(* PLC project Unnamed, Unknown Unnamed 1 *)
(* stored: creationDateTime 2024-07-23T15:43:19, modificationDateTime 2024-07-23T15:49:17 *)

PROGRAM program0
  VAR
    LocalVar0 : BOOL;
    LocalVar1 : SINT;
  END_VAR
  VAR  (* added by the conversion: wires and edge detectors of the diagram *)
    _BOOL_TO_SINT2_OUT : SINT;
    _BOOL_TO_SINT3_OUT : SINT;
  END_VAR

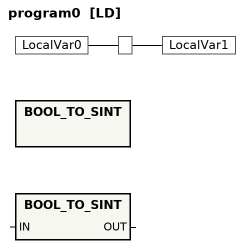
(* LD diagram, written out as Structured Text *)
LocalVar1 := ;
_BOOL_TO_SINT2_OUT := BOOL_TO_SINT();
_BOOL_TO_SINT3_OUT := BOOL_TO_SINT();
END_PROGRAM

CONFIGURATION Config0
  RESOURCE Res0 ON PLC
    TASK task0(INTERVAL := T#20ms, PRIORITY := 0);
    PROGRAM instance0 WITH task0 : program0;
  END_RESOURCE
END_CONFIGURATION
